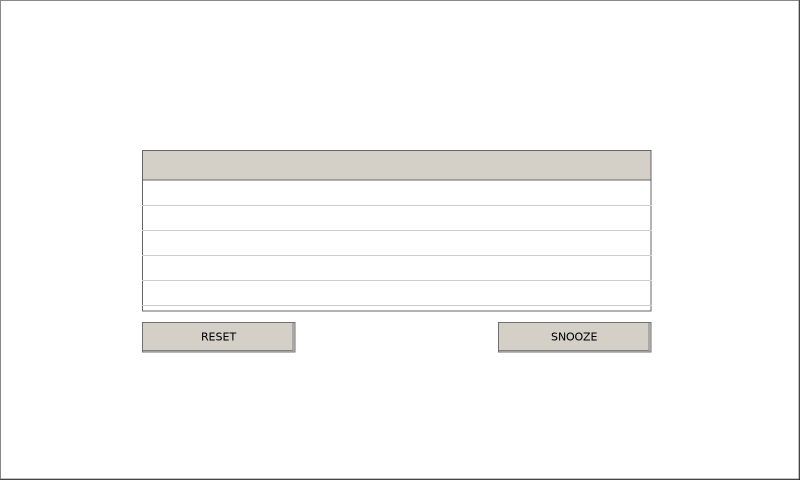
VISUALIZATION BasicMessageScreen_OLD  // 800x480
    Rectangle (0,0 800x480)
    Table (142,150 509x161), data array: Utilities_Library.GVL_Message.arActiveFaults
        p3854506369: Utilities_Library.GVL_Message.arActiveFaults[INDEX].Active
        p1892666644: Utilities_Library.GVL_Message.arActiveFaults[INDEX].FaultType
        p338671338: Utilities_Library.GVL_Message.arActiveFaults[INDEX].MessageNumber
        p2170511999: Utilities_Library.GVL_Message.arActiveFaults[INDEX].LocationNumber
        p3723444502: Utilities_Library.GVL_Message.arActiveFaults[INDEX].Discription
        p1218418051: Utilities_Library.GVL_Message.arActiveFaults[INDEX].LocationName
        p746581629: Utilities_Library.GVL_Message.arActiveFaults[INDEX].ComponentType
        p3104783080: Utilities_Library.GVL_Message.arActiveFaults[INDEX].StartTime
        p2501879983: Utilities_Library.GVL_Message.arActiveFaults[INDEX].EndTime
        p7306298: Utilities_Library.GVL_Message.arActiveFaults[INDEX].nModuleID
        p1933151965: Utilities_Library.GVL_Message.arActiveFaults[INDEX].FullFaultId
    Button (142,322 153x30), "RESET"
        tap Utilities_Library.GVL_Message.bResetFaults
    Button (498,322 153x30), "SNOOZE"
        tap Utilities_Library.GVL_Message.bCmdSnoozeMessage
END_VISUALIZATION

(* stored: Version 1.1.0.1, ProductVersion 3.1.4024.5
   Visu BasicMessageScreen_OLD: Id {30b3f472-8e76-474f-be14-9294026029ea} *)
